FUNCTION_BLOCK CNV_MDL9 (* Simple Conveyor Model for 1 Workpiece *)
  (* Standard: 61499-1; Classification: Simulation *)
  (* Version 0.0, 2004-09-20, JHC, Rockwell Automation, Simplified from CNV_MDL. *)
  (* Compiler header: package fb.rt.mva; *)
  (* Compiler Java Sun JDK 1.4.2 *)
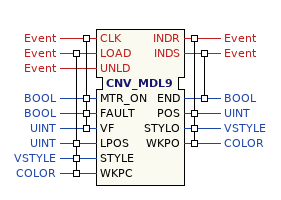
  EVENT_INPUT
    CLK WITH MTR_ON, VF, FAULT; (* Simulation Clock Event *)
    LOAD WITH STYLE, WKPC, LPOS; (* Load Workpiece if at HOME position *)
    UNLD; (* Unload Workpiece if at END position *)
  END_EVENT
  EVENT_OUTPUT
    INDR WITH POS, STYLO, WKPO; (* Change in Rendering Data *)
    INDS WITH END; (* Change in Sensor Data *)
  END_EVENT
  VAR_INPUT
    MTR_ON : BOOL; (* Motor ON command *)
    FAULT : BOOL; (* Fault Condition *)
    VF : UINT; (* Conveyor Speed in % per CLK event *)
    LPOS : UINT; (* Load Position in % of Conveyor Length *)
    STYLE : VSTYLE := NONE; (* Input Workpiece style *)
    WKPC : COLOR := yellow; (* Input Workpiece Color *)
  END_VAR
  VAR_OUTPUT
    END : BOOL; (* Workpiece at End Position *)
    POS : UINT; (* Workpiece Position in % of Conveyor Length *)
    STYLO : VSTYLE := NONE; (* Currently loaded workpiece style *)
    WKPO : COLOR := blue; (* Currently loaded workpiece color *)
  END_VAR
  ALGORITHM LOAD IN Java:
POS.value = Math.min(100,LPOS.value);
END.value = (POS.value==100)&&(STYLE.value != VSTYLE.NONE);
STYLO.value = STYLE.value;
WKPO.value = WKPC.value;
INDR.serviceEvent(this);
INDS.serviceEvent(this);
  END_ALGORITHM
  ALGORITHM UNLD IN Java:
if(STYLO.value==VSTYLE.NONE) return;
STYLO.value=VSTYLE.NONE;
END.value = false;
INDR.serviceEvent(this);
INDS.serviceEvent(this);
  END_ALGORITHM
  ALGORITHM CLK IN Java:
if(FAULT.value||END.value||!MTR_ON.value||(STYLO.value==VSTYLE.NONE)) return;
POS.value += VF.value;
if(POS.value>=120){
   POS.value=100;
   END.value=true;}
INDR.serviceEvent(this);
if(END.value) INDS.serviceEvent(this);
  END_ALGORITHM
END_FUNCTION_BLOCK
